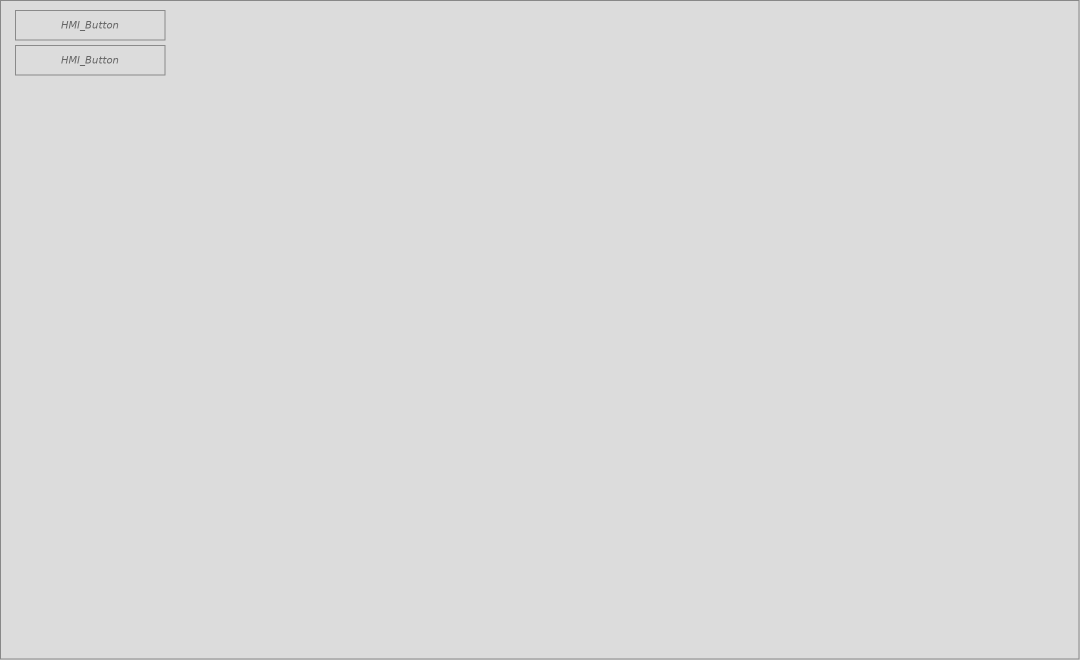
VISUALIZATION Page_PackML  // 1080x660, background image 
    Frame (15,10 150x30)
        shows HMI_Button(i_sText := 'Production', iq_stButton := GVL_Modules.g_fbHmiMachCtrlsManager.s_fbBtnReqProduction.s_stHmi)
    Frame (15,45 150x30)
        shows HMI_Button(i_sText := 'Manual', iq_stButton := GVL_Modules.g_fbHmiMachCtrlsManager.s_fbBtnReqManual.s_stHmi)
END_VISUALIZATION

(* stored: Version 1.1.0.1, ProductVersion 3.1.4026.13
   Visu Page_PackML: Id {5ee60e36-1577-47fa-97ab-d010842c2d34} *)
